Fanuc KAREL source: ko00094.KL

-- PROVISIONAL review KL for V1013-1; original PC SHA256 7db0e4be9abce0a3100ca2e891dd85bc0fd08bd9fd8f22cbacf3af78cefe8f5c
-- Incomplete behavior may be omitted. Consult companion uncertainty JSON. Do not deploy.
PROGRAM KO00094
%NOLOCKGROUP
BEGIN
  -- UNRESOLVED_PC offsets 5-12; opcodes 9D,23
  -- UNRESOLVED_PC offsets 17-69; opcodes 27,27,49,7E,AD,27,49,7E,AD,22,31,7E,4A
  -- UNRESOLVED_PC offsets 74-78; opcodes 7F
END KO00094
